{attribute addProperty BoxType "ATH2050-0500-0022"}
{attribute addProperty Id "CC_InputsAT %I*CC_Inputs_9818D8D8256320CC_OutputsAT %Q*CC_Outputs_AA78E99F256320WcStateAT %I*WcState_F855686C1620InfoDataAT %I*InfoData_0BDED7BF144180"}
{attribute addProperty CRC "2581212370"}
{attribute addProperty SizeInBites "672"}
{attribute addProperty SizeInBytes "84"}
TYPE ATH2050_9506A482 :
STRUCT
	{attribute addProperty Name "CC_Inputs"}
	CC_Inputs : CC_Inputs_9818D8D8;
	{attribute addProperty Name "CC_Outputs"}
	CC_Outputs : CC_Outputs_AA78E99F;
	{attribute addProperty Name "WcState"}
	WcState : WcState_F855686C;
	{attribute addProperty Name "InfoData"}
	InfoData : InfoData_0BDED7BF;
END_STRUCT
END_TYPE

(* stored: Version 1.2.0.0, ProductVersion 3.1.4024.9
   DUT ATH2050_9506A482: Id {5da6c75a-6403-4e34-8690-547170722ff7} *)
